FUNCTION_BLOCK PAEActValve EXTENDS PAEActuator1way
VAR_INPUT
END_VAR
VAR_OUTPUT
END_VAR
VAR
END_VAR

METHOD FB_init : BOOL
VAR_INPUT
	bInitRetains : BOOL; // if TRUE, the retain variables are initialized (warm start / cold start)
	bInCopyCode : BOOL;  // if TRUE, the instance afterwards gets moved into the copy code (online change)
	parent : IACComponent;
END_VAR
END_METHOD

END_FUNCTION_BLOCK

(* stored: Version 1.1.0.1, ProductVersion 3.1.4024.6
   POU PAEActValve: Id {2e9e0893-b9af-4ab8-aa78-98b7c83fff2e}, SpecialFunc None
   Method FB_init: Id {27610ff8-8d86-4033-b8ad-e2c8f1a9957e} *)
